SUBAPPLICATION Uebung_034b (* LONG_PRESS_HOLD-Eingang auf PWM Ausgang *)
  (* Standard: 61499-2; Description: Copyright (c) 2023 Meisterschulen am Ostbahnhof This program and the accompanying materials are made available under the terms of the Eclipse Public License 2.0 which is available at https://www.eclipse.org/legal/epl-2.0/ SPDX-License-Identifier: EPL-2.0 *)
  (* Version 1.0, 2023-10-23, Franz Höpfinger, Meisterschulen am Ostbahnhof *)
  IMPORT logiBUS::io::DI::logiBUS_DI;
  IMPORT logiBUS::io::DI::logiBUS_DI_Events;
  IMPORT logiBUS::io::DQ::logiBUS_DO;
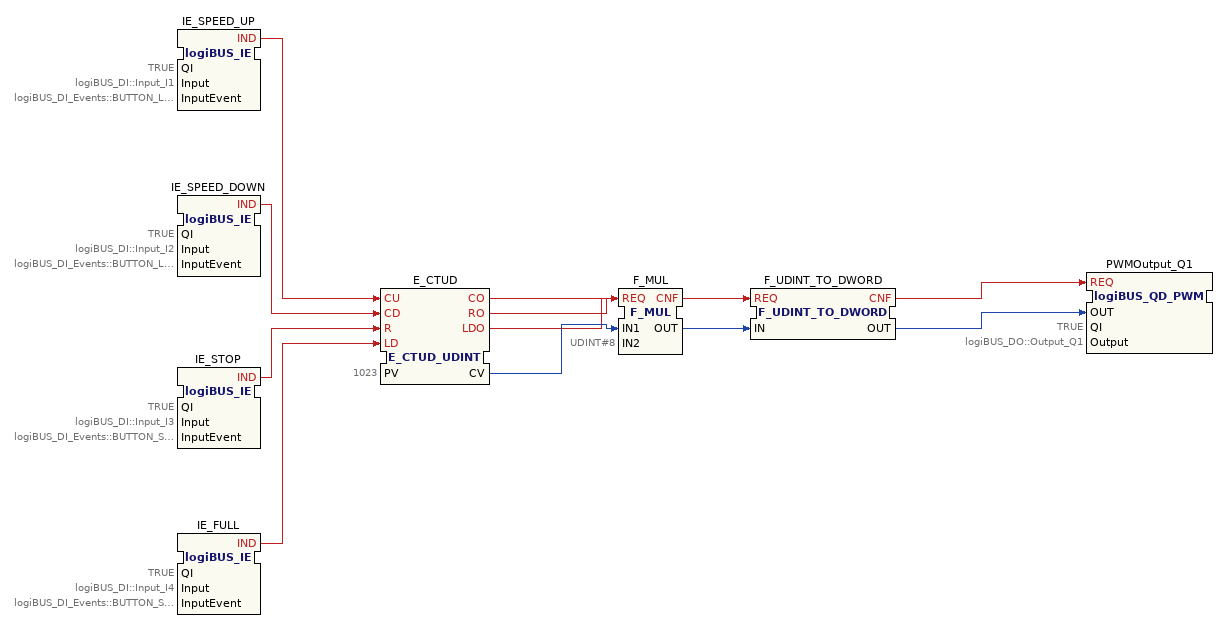
  FBS
    PWMOutput_Q1 : logiBUS::io::DQ::logiBUS_QD_PWM(QI := TRUE, Output := logiBUS_DO::Output_Q1);
    IE_SPEED_UP : logiBUS::io::DI::logiBUS_IE(QI := TRUE, Input := logiBUS_DI::Input_I1, InputEvent := logiBUS_DI_Events::BUTTON_LONG_PRESS_HOLD);
    IE_SPEED_DOWN : logiBUS::io::DI::logiBUS_IE(QI := TRUE, Input := logiBUS_DI::Input_I2, InputEvent := logiBUS_DI_Events::BUTTON_LONG_PRESS_HOLD);
    E_CTUD : iec61499::events::E_CTUD_UDINT(PV := 1023);
    F_UDINT_TO_DWORD : iec61131::conversion::F_UDINT_TO_DWORD;
    IE_STOP : logiBUS::io::DI::logiBUS_IE(QI := TRUE, Input := logiBUS_DI::Input_I3, InputEvent := logiBUS_DI_Events::BUTTON_SINGLE_CLICK);
    IE_FULL : logiBUS::io::DI::logiBUS_IE(QI := TRUE, Input := logiBUS_DI::Input_I4, InputEvent := logiBUS_DI_Events::BUTTON_SINGLE_CLICK);
    F_MUL : iec61131::arithmetic::F_MUL(IN2 := UDINT#8);
  END_FBS
  EVENT_CONNECTIONS
    E_CTUD.CO TO F_MUL.REQ;
    E_CTUD.RO TO F_MUL.REQ;
    IE_SPEED_UP.IND TO E_CTUD.CU;
    IE_SPEED_DOWN.IND TO E_CTUD.CD;
    IE_STOP.IND TO E_CTUD.R;
    IE_FULL.IND TO E_CTUD.LD;
    E_CTUD.LDO TO F_MUL.REQ;
    F_UDINT_TO_DWORD.CNF TO PWMOutput_Q1.REQ;
    F_MUL.CNF TO F_UDINT_TO_DWORD.REQ;
  END_CONNECTIONS
  DATA_CONNECTIONS
    E_CTUD.CV TO F_MUL.IN1;
    F_UDINT_TO_DWORD.OUT TO PWMOutput_Q1.OUT;
    F_MUL.OUT TO F_UDINT_TO_DWORD.IN;
  END_CONNECTIONS
END_SUBAPPLICATION
